{attribute 'linkalways'} 
{attribute 'no_explicit_call' := 'This FB is a CLASS and must be accessed using methods or properties'}
{attribute 'enable_dynamic_creation'}
FUNCTION_BLOCK Node_F_VN_DrawRotatedRectangle EXTENDS VisionNode
VAR
    stRectangle : _TcVnRotatedRectangle;
    ipDestImage : _ITcVnImage;
    aColor : _TcVnVector4_LREAL;
    nThickness : _DINT(1);
    hrPrev : _HRESULT(S_OK);
	hresult : _HRESULT(S_OK);
END_VAR

METHOD PUBLIC  Clone : I_Node
VAR
	pNode : POINTER TO Node_F_VN_DrawRotatedRectangle;
END_VAR
pNode := __NEW(Node_F_VN_DrawRotatedRectangle);
Clone := pNode^;
END_METHOD

METHOD FB_init : BOOL
VAR_INPUT
	bInitRetains : BOOL; // if TRUE, the retain variables are initialized (warm start / cold start)
	bInCopyCode : BOOL;  // if TRUE, the instance afterwards gets moved into the copy code (online change)
END_VAR
AddInput('stRectangle', stRectangle);
AddInput('ipDestImage', ipDestImage);
AddInput('aColor', aColor);
AddParameter('nThickness', nThickness);
AddInput('hrPrev', hrPrev);
AddOutput('ipDestImage', ipDestImage);
AddOutput('hresult',hresult);
END_METHOD

METHOD PROTECTED OnExecute
hresult.Value := F_VN_DrawRotatedRectangle(
    stRectangle := stRectangle.Value,
	ipDestImage := ipDestImage.Value,
    aColor := aColor.Value,
    nThickness := nThickness.Value,
	hrPrev:= hrPrev.Value);
END_METHOD

METHOD PUBLIC PreExecutionCheck
VAR_INPUT
	Check : I_PreExecutionChecks;
END_VAR
Check.IsTrue(ipDestImage.IsValid, 'ipDestImage must contain an image');
Check.IsTrue(nThickness.Value <> 0, 'nThickness must be non-zero');
END_METHOD

END_FUNCTION_BLOCK

(* stored: Version 1.1.0.1, ProductVersion 3.1.4024.15
   POU Node_F_VN_DrawRotatedRectangle: Id {b0f75431-6f75-09b9-0ba7-077d9dda4bc4}, SpecialFunc None
   Folder Constructor: Id {9167fd85-4a87-01ad-3a39-43469fac4806}
   Method Clone: Id {68b5c734-51f2-0b76-178f-5f49dc34999a}
   Method FB_init: Id {bc676d8f-1d95-0de6-135c-4d6dc1ac1c68}
   Method OnExecute: Id {2162ba4a-bb2d-04a5-27f8-16d80d9603cc}
   Method PreExecutionCheck: Id {bfa26380-1aa8-0200-3a42-59ba429011e3} *)
